# EPICS substitutions: apps/jscalerApp/Db/jscalers_TDCFTOF3_TRIG.substitutions
file "db/jscaler_channel.db" {
pattern { CrNo,CrName,Sl,Ch,Det,Sys,Element,CScode,Thresh,Mode,Counts }
{ "05","TDCFTOF3","20","15","TRIG","DISC","SEC3_F00","5125","15","271","15" }
}
